FUNCTION_BLOCK Performance1 (* Composite Function Block Type *)
  (* Standard: 61499-2 *)
  (* Version 1.0, 2020-12-26, jetbrains *)
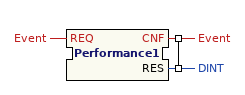
  EVENT_INPUT
    REQ; (* Normal Execution Request *)
  END_EVENT
  EVENT_OUTPUT
    CNF WITH RES; (* Execution Confirmation *)
  END_EVENT
  VAR_OUTPUT
    RES : DINT; (* Output event qualifier *)
  END_VAR
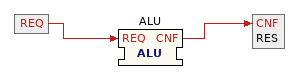
  FBS
    ALU : ALU;
  END_FBS
  EVENT_CONNECTIONS
    REQ TO ALU.REQ;
    ALU.CNF TO CNF;
  END_CONNECTIONS
END_FUNCTION_BLOCK
